(* IEC 61131-3 sources: unipi_neuron_test/mervis_test_project/bin, 2 files *)

(* ---- 0.st ---- *)
namespace $HW_hidden$

var_global
	$1Wire.1W-Thermometer.Temperature$ : $int$ ;
	$tmp_real$ : $real$ ;
	$1Wire.1W-Thermometer.Temperature.transformation$ : $lib$.$core$.$v1_0$.$linear$ := ($k$ := 0.0625);
end_var

program f_transform
		$tmp_real$ := $1Wire.1W-Thermometer.Temperature.transformation$.Forward(in := $1Wire.1W-Thermometer.Temperature$);

		$hw$.$1w-thermometer_temperature$ := $tmp_real$;

end_program
program r_transform
end_program
program init_transform

end_program
program finish_transform

end_program
end_namespace

(* ---- main_a5bb432f-6ef2-4d12-8e62-5717f2a301f1.generated.st ---- *)
program main
var
	//63eded8e-9a38-42f1-8559-8eaf5c5a8721
	$B36_PID_Controller$ : Lib.Core.V1_0.B36_PID_Controller;
end_var

	//c71d12bf-3ef0-48ec-b731-24495089412b

	//df84dbe9-cb23-492a-8a4e-3b4b70fa9d40

	//63eded8e-9a38-42f1-8559-8eaf5c5a8721
	$B36_PID_Controller$($x$ := $hw$.$1W-Thermometer_Convert_commblock$, $w$ := $Desired_temperature$);
	//68940fa5-7090-44f1-a0f9-6276dc064282
	$hw$.$Neuron S10x_DO_1.01$ := $B36_PID_Controller$.$Out$
end_program
